(*
	Estados DO ciclo automático DO simulado de certificação (Exercício 07).

    PARADO           -> máquina ociosa, aguardando comando de ligar ciclo.
    POSICIONA_FUSO    -> passo A: leva o fuso para a posição de repouso (5 mm).
    POSICIONA_MESA    -> passo B: garante que a mesa esteja numa posição de produto.
    AVANCA_FERRAMENTA -> passo C (parte 1): avança o fuso até 40 mm.
    AGUARDA_OPERACAO  -> passo C (parte 2): aguarda 1s na posição de trabalho.
    RECUA_FERRAMENTA  -> passo C (parte 3): recua o fuso de volta a 5 mm.
    GIRA_MESA         -> passo D: indexa a mesa para a próxima posição de produto.
*)
TYPE E_EstadoCicloAutomatico :
(
    PARADO,
    POSICIONA_FUSO,
    POSICIONA_MESA,
    AVANCA_FERRAMENTA,
    AGUARDA_OPERACAO,
    RECUA_FERRAMENTA,
    GIRA_MESA
);
END_TYPE

(* stored: Version 1.1.0.1
   DUT E_EstadoCicloAutomatico: Id {a1b2c3d4-0001-4002-8002-000000000006} *)
